// TIA Portal V17 export
// export: Created 2022-02-03T14:45:11.5284152Z, ExportSetting WithDefaults, DisplayName Totally Integrated Automation Portal, DisplayVersion V17, DisplayName TIA Portal Openness, DisplayVersion V17, DisplayName TIA Portal Version Control Interface, DisplayVersion V17, DisplayName SINAMICS Startdrive Advanced, DisplayVersion V17, DisplayName SINAMICS Startdrive G130, G150, S120, S150, SINAMICS MV, S210, DisplayVersion V17, DisplayName SINAMICS Startdrive G110M, G120, G120C, G120D, G120P, G115D, DisplayVersion V17, DisplayName STEP 7 Professional, DisplayVersion V17, DisplayName STEP 7 Safety, DisplayVersion V17, DisplayName WinCC Advanced, DisplayVersion V17
ORGANIZATION_BLOCK "MainSignal"   // OB124, LAD, ProgramCycle
TITLE = "Main Program Sweep (Cycle)"
VERSION : 0.1
// stored: AutoNumber true, IsIECCheckEnabled false, SetENOAutomatically false
   VAR_INPUT
      Initial_Call : Bool;   // Initial call of this OB
      Remanence : Bool;   // =True, if remanent data are available
   END_VAR
BEGIN

REGION Network 1
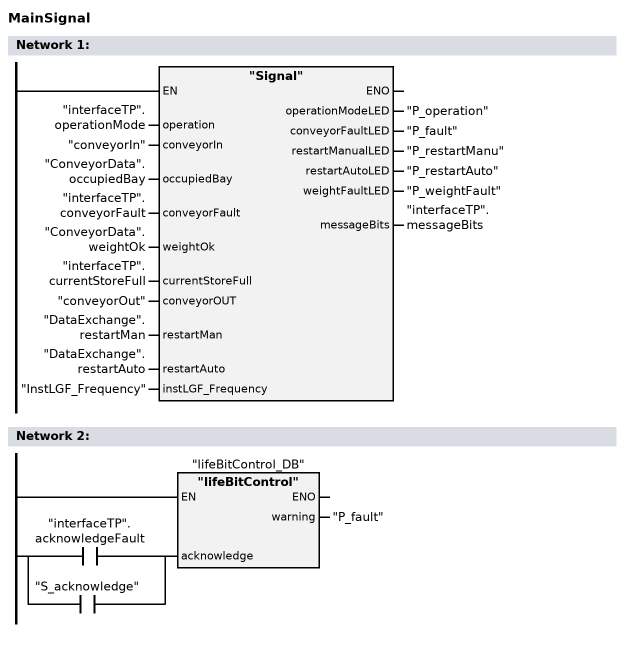
   RUNG wire#powerrail
      "Signal"(operation := "interfaceTP".operationMode, conveyorIn := "conveyorIn", occupiedBay := "ConveyorData".occupiedBay, conveyorFault := "interfaceTP".conveyorFault, weightOk := "ConveyorData".weightOk, currentStoreFull := "interfaceTP".currentStoreFull, conveyorOUT := "conveyorOut", restartMan := "DataExchange".restartMan, restartAuto := "DataExchange".restartAuto, instLGF_Frequency := "InstLGF_Frequency", operationModeLED => "P_operation", conveyorFaultLED => "P_fault", restartManualLED => "P_restartManu", restartAutoLED => "P_restartAuto", weightFaultLED => "P_weightFault", messageBits => "interfaceTP".messageBits)
   END_RUNG
   // the same network as SCL:
   "Signal"(operation := "interfaceTP".operationMode,
            conveyorIn := "conveyorIn",
            occupiedBay := "ConveyorData".occupiedBay,
            conveyorFault := "interfaceTP".conveyorFault,
            weightOk := "ConveyorData".weightOk,
            currentStoreFull := "interfaceTP".currentStoreFull,
            conveyorOUT := "conveyorOut",
            restartMan := "DataExchange".restartMan,
            restartAuto := "DataExchange".restartAuto,
            instLGF_Frequency := "InstLGF_Frequency",
            operationModeLED => "P_operation",
            conveyorFaultLED => "P_fault",
            restartManualLED => "P_restartManu",
            restartAutoLED => "P_restartAuto",
            weightFaultLED => "P_weightFault",
            messageBits => "interfaceTP".messageBits);
END_REGION

REGION Network 2
   RUNG wire#powerrail
      "lifeBitControl_DB"(acknowledge := wire#w1, warning => "P_fault")
   END_RUNG
   RUNG wire#powerrail
      Contact( "interfaceTP".acknowledgeFault )
   END_RUNG wire#w1
   RUNG wire#powerrail
      Contact( "S_acknowledge" )
   END_RUNG wire#w1
   // the same network as SCL:
   "lifeBitControl_DB"(acknowledge := "interfaceTP".acknowledgeFault OR "S_acknowledge", warning => "P_fault");   // "lifeBitControl"
END_REGION
END_ORGANIZATION_BLOCK
